// TIA Portal V20 export
TYPE "typeAxisInterlockpermit"
// stored: Access Published
   STRUCT
      general : Bool;
      jogForward : Bool;
      jogBackward : Bool;
   END_STRUCT;
END_TYPE
